# EPICS StreamDevice protocol: ipApp/Db/Digitel_stream.proto
# Digitel_stream.proto

# Stream protocol file for Digital 500/1500 ion pump controllers

# Mark Rivers
# May 16, 2024

ExtraInput = Ignore;
ReadTimeout = 1000;

readVI {
   out "RD";
   in "%*s";
   in "%*9c%fV%(\$1_Current)fI%*7c";
}
